FUNCTION F_ArchRadToCstcaAngle : UINT
VAR_INPUT
    theta : LREAL;
END_VAR
VAR CONSTANT
    TWO_PI : LREAL := 6.2831853071795864769;
END_VAR
VAR
    wrapped : LREAL;
    counts  : DINT;
END_VAR

wrapped := F_ArchWrap2Pi(theta);
counts := LREAL_TO_DINT(wrapped / TWO_PI * 65536.0);
IF counts >= 65536 THEN
    counts := counts - 65536;
ELSIF counts < 0 THEN
    counts := counts + 65536;
END_IF
F_ArchRadToCstcaAngle := DINT_TO_UINT(counts);

END_FUNCTION

(* stored: Version 1.1.0.1, ProductVersion 3.1.4024.12
   POU F_ArchRadToCstcaAngle: Id {9f95b821-e6f9-4e51-98dd-900047a02002}, SpecialFunc None *)
